FUNCTION alg_a_transfer2pickpos : BOOL
VAR_INPUT
	state: STATE;
END_VAR

alg_a_transfer2pickpos := FALSE;

END_FUNCTION

(* stored: Version 1.1.0.1, ProductVersion 3.1.4022.18
   POU alg_a_transfer2pickpos: Id {20fef1de-9a0b-4aab-b8d6-089cc64e7185}, SpecialFunc None *)
